Fanuc KAREL source: kt00478.KL

-- PROVISIONAL review KL for V1013-1; original PC SHA256 cadf2d4eef8ce2894a1c935fb3ea436953bb55ba39593ed17df525cc49f06498
-- Incomplete behavior may be omitted. Consult companion uncertainty JSON. Do not deploy.
PROGRAM KT00478
%NOLOCKGROUP
VAR
  OUT : BOOLEAN
-- UNRESOLVED_DECL P1 type=000101
-- UNRESOLVED_DECL P2 type=000102
BEGIN
  -- UNRESOLVED_PC offsets 5-20; opcodes 2E,22,32,35
  -- UNRESOLVED_PC offsets 25-53; opcodes 49,49,7E,AC,23
  -- UNRESOLVED_PC offsets 58-62; opcodes 7F
END KT00478
